INTERFACE I_Shape

END_INTERFACE

(* stored: Version 1.1.0.1, ProductVersion 3.1.4024.13
   Itf I_Shape: Id {b93cf4af-7d3c-436b-9d9b-fbf93c1274ed} *)
